// TIA Portal V21 export
VAR_GLOBAL   // PLC tag table "UnitaDiMisura_MulSottomul"
END_VAR
VAR_GLOBAL CONSTANT   // user constants
   Um_MulSottomul_Metri_µm : Int := 1;
   Um_MulSottomul_Metri_mm : Int := 2;
   Um_MulSottomul_Metri_cm : Int := 3;
   Um_MulSottomul_Metri_dm : Int := 4;
   Um_MulSottomul_Metri_m : Int := 5;
   Um_MulSottomul_Metri_dam : Int := 6;
   Um_MulSottomul_Metri_hm : Int := 7;
   Um_MulSottomul_Metri_km : Int := 8;
   Um_MulSottomul_Metri_Megametro : Int := 9;
   Um_MulSottomul_Pollice_Pollice : Int := 5;
   "Um_MulSottomul_Pollice_3/4Pollice" : Int := 4;
   "Um_MulSottomul_Pollice_1/2Pollice" : Int := 3;
   "Um_MulSottomul_Pollice_1/4Pollice" : Int := 2;
   "Um_MulSottomul_Pollice_1/8Pollice" : Int := 1;
   "Um_MulSottomul_Percentuale_1%" : Int := 5;
   Um_MulSottomul_Piedi_Piede : Int := 5;
   "Um_MulSottomul_°C" : Int := 5;
   "Um_MulSottomul_°F" : Int := 5;
   Um_MulSottomul_K : Int := 5;
   Um_MulSottomul_Portata_MetriCubih : Int := 5;
   Um_MulSottomul_Portata_LitriMin : Int := 5;
   Um_MulSottomul_Bar_bar : Int := 5;
   Um_MulSottomul_Bar_Millibar : Int := 2;
   Um_MulSottomul_Bar_Centibar : Int := 3;
   Um_MulSottomul_Bar_decibar : Int := 4;
   Um_MulSottomul_Portata_Litrih : Int := 6;
   "Um_MulSottomul_mg/l_mg/l" : Int := 5;
END_VAR
